PROGRAM MAIN
VAR
	boolTo_TestSuit : BOOL_TO_TestSuit;
	byteTo_TestSuit : BYTE_TO_TestSuit;
	dateTo_TestSuit : DATE_TO_TestSuit;
END_VAR

TcUnit.RUN();

END_PROGRAM

(* stored: Version 1.1.0.1, ProductVersion 3.1.4024.12
   POU MAIN: Id {7c22aba4-4a89-069c-18cd-1d4a5752fff2}, SpecialFunc None *)
